Fanuc KAREL source: kb00129.KL

-- PROVISIONAL review KL for V940-1; original PC SHA256 13cc67890a1dd206eab6891048306e07bdca6f63cc7f9123b95e5c558c03065e
-- Incomplete behavior may be omitted. Consult companion uncertainty JSON. Do not deploy.
PROGRAM KB00129
%NOLOCKGROUP
BEGIN
  -- V9_ZERO_TABLE_METADATA_HINT layout=0002_ascii; no indexed target words; source/name/runtime held
  -- UNRESOLVED_PC offsets 5-14; opcodes 3F,75
  -- UNRESOLVED_PC offsets 19-26; opcodes 9D,23
  -- UNRESOLVED_PC offsets 31-38; opcodes 9D,23
  -- UNRESOLVED_PC offsets 43-50; opcodes 9D,23
  -- UNRESOLVED_PC offsets 55-85; opcodes 27,22,2A,22,22,22,31
  -- UNRESOLVED_PC offsets 90-94; opcodes 7F
END KB00129
